PROGRAM OUTPUTS
VAR
	C6_K1_SAFETY_CONTACTOR AT %Q*: BOOL; // 
	C6_K2_SAFETY_CONTACTOR AT %Q*: BOOL; // 
	C7_K1_SAFETY_CONTACTOR AT %Q*: BOOL; // 
	C7_K2_SAFETY_CONTACTOR AT %Q*: BOOL; // 	



KIRK_BIT: BOOL;
BTEST :BOOL;
	
//GL4: sConveyor;
	

//GL5A:sConveyor;
	
	
//GL5B: sConveyor;
//GL6: sConveyor;
//GL7: sConveyor;
//GL8: sConveyor;
//GL9: sConveyor;
	
END_VAR

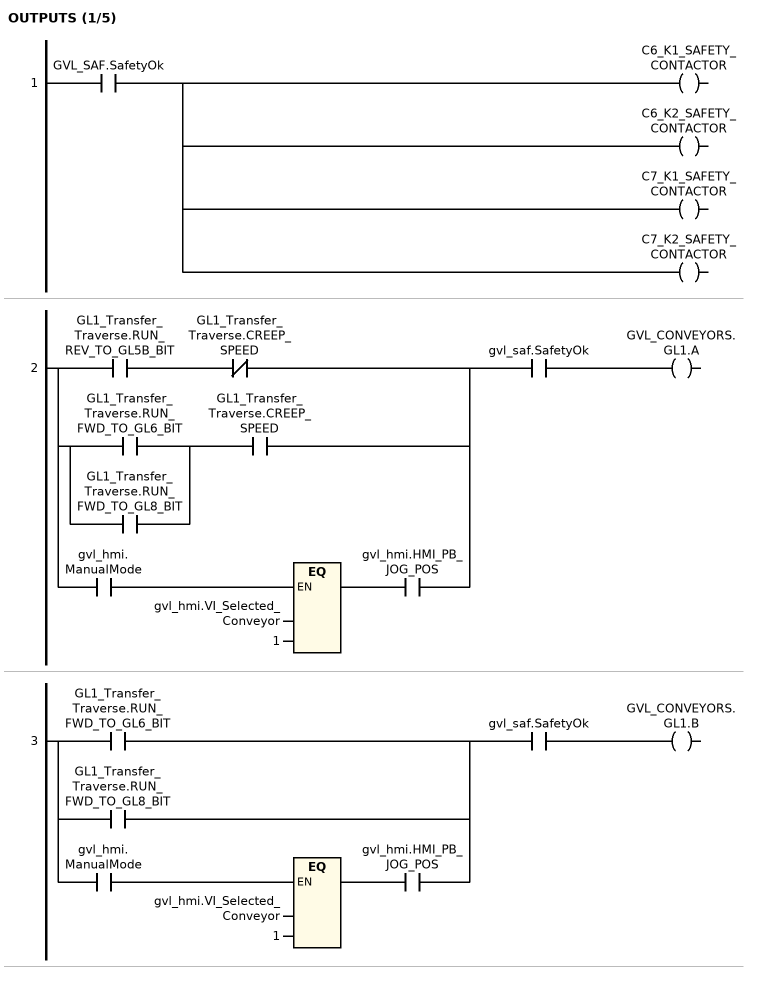
// NETWORK 1
C6_K1_SAFETY_CONTACTOR := GVL_SAF.SafetyOk;
C6_K2_SAFETY_CONTACTOR := GVL_SAF.SafetyOk;
C7_K1_SAFETY_CONTACTOR := GVL_SAF.SafetyOk;
C7_K2_SAFETY_CONTACTOR := GVL_SAF.SafetyOk;

// NETWORK 2
GVL_CONVEYORS.GL1.A := (GL1_Transfer_Traverse.RUN_REV_TO_GL5B_BIT AND NOT GL1_Transfer_Traverse.CREEP_SPEED OR (GL1_Transfer_Traverse.RUN_FWD_TO_GL6_BIT OR GL1_Transfer_Traverse.RUN_FWD_TO_GL8_BIT) AND GL1_Transfer_Traverse.CREEP_SPEED OR (gvl_hmi.ManualMode AND gvl_hmi.VI_Selected_Conveyor = 1) AND gvl_hmi.HMI_PB_JOG_POS) AND gvl_saf.SafetyOk;

// NETWORK 3
GVL_CONVEYORS.GL1.B := (GL1_Transfer_Traverse.RUN_FWD_TO_GL6_BIT OR GL1_Transfer_Traverse.RUN_FWD_TO_GL8_BIT OR (gvl_hmi.ManualMode AND gvl_hmi.VI_Selected_Conveyor = 1) AND gvl_hmi.HMI_PB_JOG_POS) AND gvl_saf.SafetyOk;

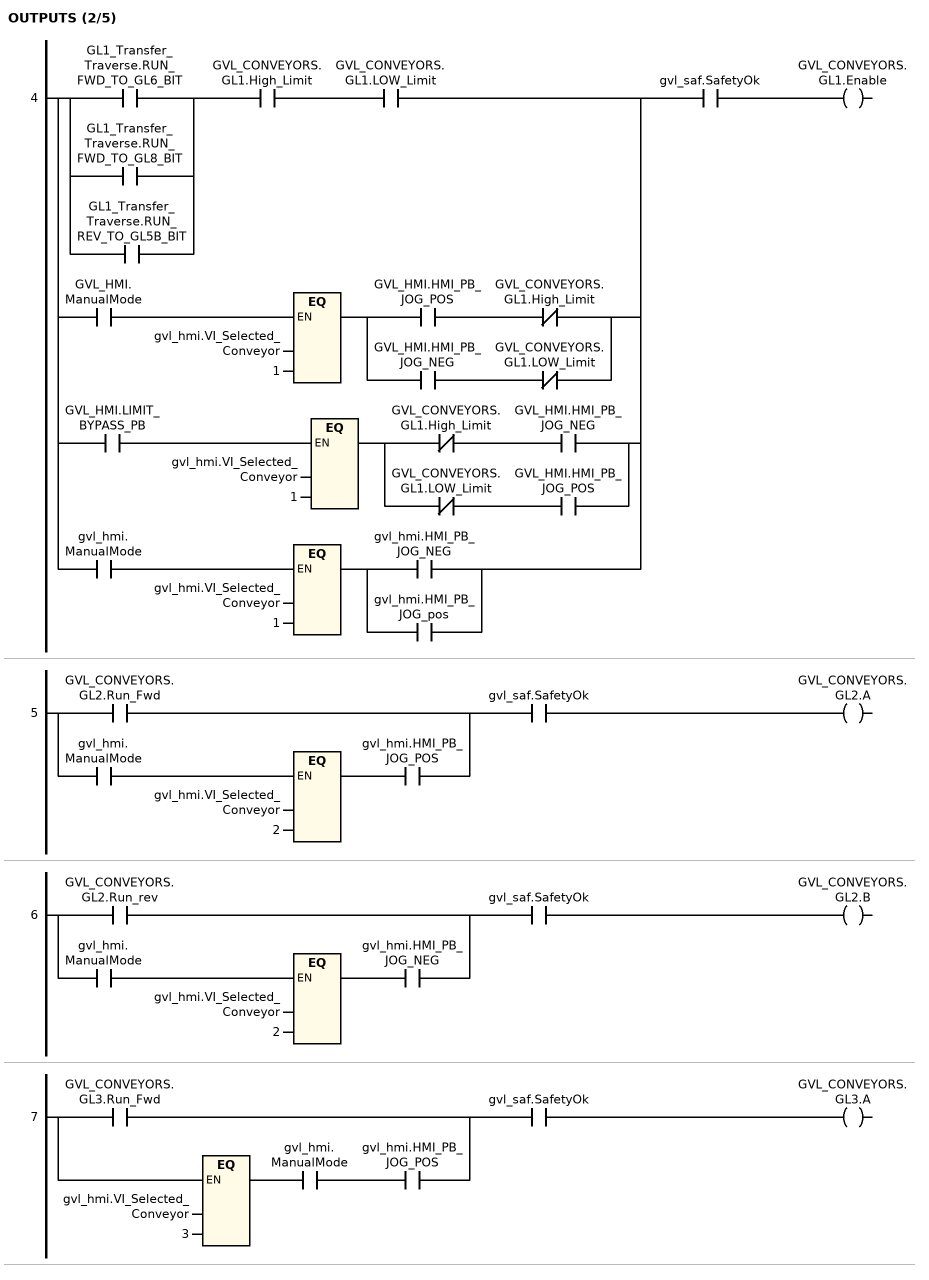
// NETWORK 4
GVL_CONVEYORS.GL1.Enable := ((GL1_Transfer_Traverse.RUN_FWD_TO_GL6_BIT OR GL1_Transfer_Traverse.RUN_FWD_TO_GL8_BIT OR GL1_Transfer_Traverse.RUN_REV_TO_GL5B_BIT) AND GVL_CONVEYORS.GL1.High_Limit AND GVL_CONVEYORS.GL1.LOW_Limit OR (GVL_HMI.ManualMode AND gvl_hmi.VI_Selected_Conveyor = 1) AND (GVL_HMI.HMI_PB_JOG_POS AND NOT GVL_CONVEYORS.GL1.High_Limit OR GVL_HMI.HMI_PB_JOG_NEG AND NOT GVL_CONVEYORS.GL1.LOW_Limit) OR (GVL_HMI.LIMIT_BYPASS_PB AND gvl_hmi.VI_Selected_Conveyor = 1) AND (NOT GVL_CONVEYORS.GL1.High_Limit AND GVL_HMI.HMI_PB_JOG_NEG OR NOT GVL_CONVEYORS.GL1.LOW_Limit AND GVL_HMI.HMI_PB_JOG_POS) OR (gvl_hmi.ManualMode AND gvl_hmi.VI_Selected_Conveyor = 1) AND (gvl_hmi.HMI_PB_JOG_NEG OR gvl_hmi.HMI_PB_JOG_pos)) AND gvl_saf.SafetyOk;

// NETWORK 5
GVL_CONVEYORS.GL2.A := (GVL_CONVEYORS.GL2.Run_Fwd OR (gvl_hmi.ManualMode AND gvl_hmi.VI_Selected_Conveyor = 2) AND gvl_hmi.HMI_PB_JOG_POS) AND gvl_saf.SafetyOk;

// NETWORK 6
GVL_CONVEYORS.GL2.B := (GVL_CONVEYORS.GL2.Run_rev OR (gvl_hmi.ManualMode AND gvl_hmi.VI_Selected_Conveyor = 2) AND gvl_hmi.HMI_PB_JOG_NEG) AND gvl_saf.SafetyOk;

// NETWORK 7
GVL_CONVEYORS.GL3.A := (GVL_CONVEYORS.GL3.Run_Fwd OR gvl_hmi.VI_Selected_Conveyor = 3 AND gvl_hmi.ManualMode AND gvl_hmi.HMI_PB_JOG_POS) AND gvl_saf.SafetyOk;

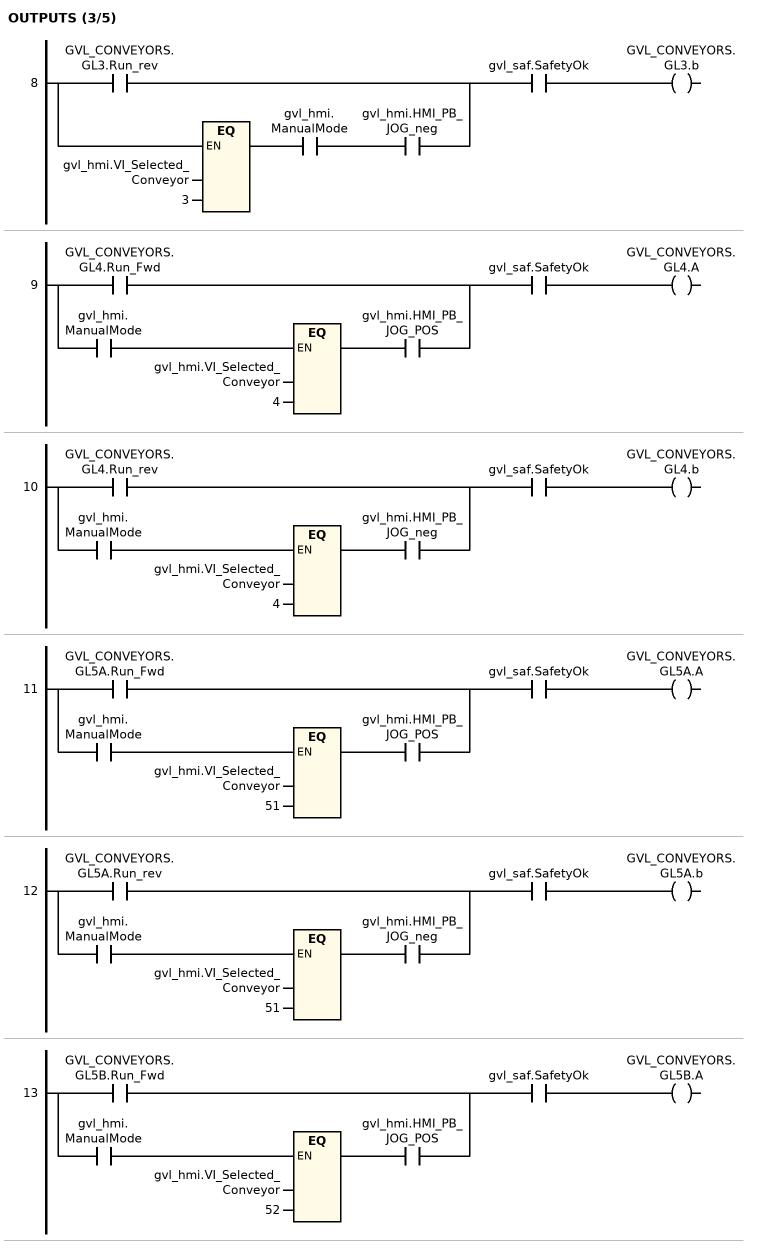
// NETWORK 8
GVL_CONVEYORS.GL3.b := (GVL_CONVEYORS.GL3.Run_rev OR gvl_hmi.VI_Selected_Conveyor = 3 AND gvl_hmi.ManualMode AND gvl_hmi.HMI_PB_JOG_neg) AND gvl_saf.SafetyOk;

// NETWORK 9
GVL_CONVEYORS.GL4.A := (GVL_CONVEYORS.GL4.Run_Fwd OR (gvl_hmi.ManualMode AND gvl_hmi.VI_Selected_Conveyor = 4) AND gvl_hmi.HMI_PB_JOG_POS) AND gvl_saf.SafetyOk;

// NETWORK 10
GVL_CONVEYORS.GL4.b := (GVL_CONVEYORS.GL4.Run_rev OR (gvl_hmi.ManualMode AND gvl_hmi.VI_Selected_Conveyor = 4) AND gvl_hmi.HMI_PB_JOG_neg) AND gvl_saf.SafetyOk;

// NETWORK 11
GVL_CONVEYORS.GL5A.A := (GVL_CONVEYORS.GL5A.Run_Fwd OR (gvl_hmi.ManualMode AND gvl_hmi.VI_Selected_Conveyor = 51) AND gvl_hmi.HMI_PB_JOG_POS) AND gvl_saf.SafetyOk;

// NETWORK 12
GVL_CONVEYORS.GL5A.b := (GVL_CONVEYORS.GL5A.Run_rev OR (gvl_hmi.ManualMode AND gvl_hmi.VI_Selected_Conveyor = 51) AND gvl_hmi.HMI_PB_JOG_neg) AND gvl_saf.SafetyOk;

// NETWORK 13
GVL_CONVEYORS.GL5B.A := (GVL_CONVEYORS.GL5B.Run_Fwd OR (gvl_hmi.ManualMode AND gvl_hmi.VI_Selected_Conveyor = 52) AND gvl_hmi.HMI_PB_JOG_POS) AND gvl_saf.SafetyOk;

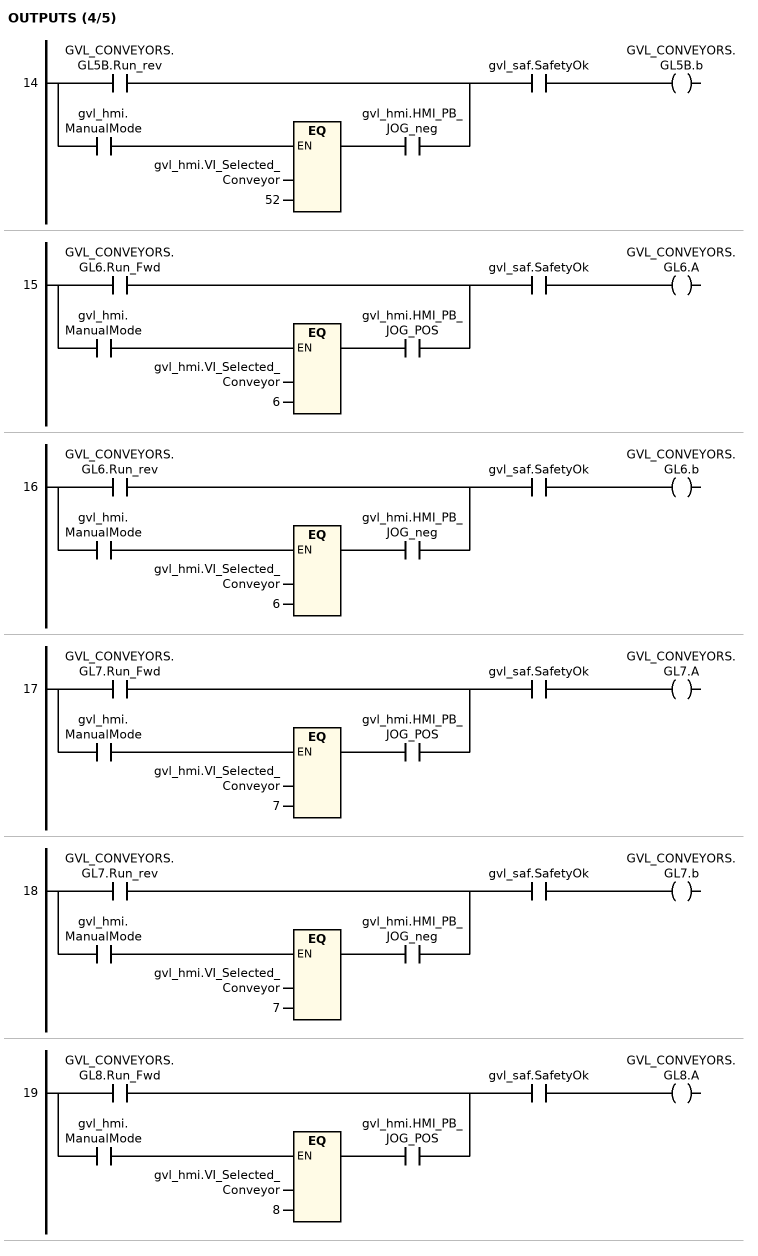
// NETWORK 14
GVL_CONVEYORS.GL5B.b := (GVL_CONVEYORS.GL5B.Run_rev OR (gvl_hmi.ManualMode AND gvl_hmi.VI_Selected_Conveyor = 52) AND gvl_hmi.HMI_PB_JOG_neg) AND gvl_saf.SafetyOk;

// NETWORK 15
GVL_CONVEYORS.GL6.A := (GVL_CONVEYORS.GL6.Run_Fwd OR (gvl_hmi.ManualMode AND gvl_hmi.VI_Selected_Conveyor = 6) AND gvl_hmi.HMI_PB_JOG_POS) AND gvl_saf.SafetyOk;

// NETWORK 16
GVL_CONVEYORS.GL6.b := (GVL_CONVEYORS.GL6.Run_rev OR (gvl_hmi.ManualMode AND gvl_hmi.VI_Selected_Conveyor = 6) AND gvl_hmi.HMI_PB_JOG_neg) AND gvl_saf.SafetyOk;

// NETWORK 17
GVL_CONVEYORS.GL7.A := (GVL_CONVEYORS.GL7.Run_Fwd OR (gvl_hmi.ManualMode AND gvl_hmi.VI_Selected_Conveyor = 7) AND gvl_hmi.HMI_PB_JOG_POS) AND gvl_saf.SafetyOk;

// NETWORK 18
GVL_CONVEYORS.GL7.b := (GVL_CONVEYORS.GL7.Run_rev OR (gvl_hmi.ManualMode AND gvl_hmi.VI_Selected_Conveyor = 7) AND gvl_hmi.HMI_PB_JOG_neg) AND gvl_saf.SafetyOk;

// NETWORK 19
GVL_CONVEYORS.GL8.A := (GVL_CONVEYORS.GL8.Run_Fwd OR (gvl_hmi.ManualMode AND gvl_hmi.VI_Selected_Conveyor = 8) AND gvl_hmi.HMI_PB_JOG_POS) AND gvl_saf.SafetyOk;

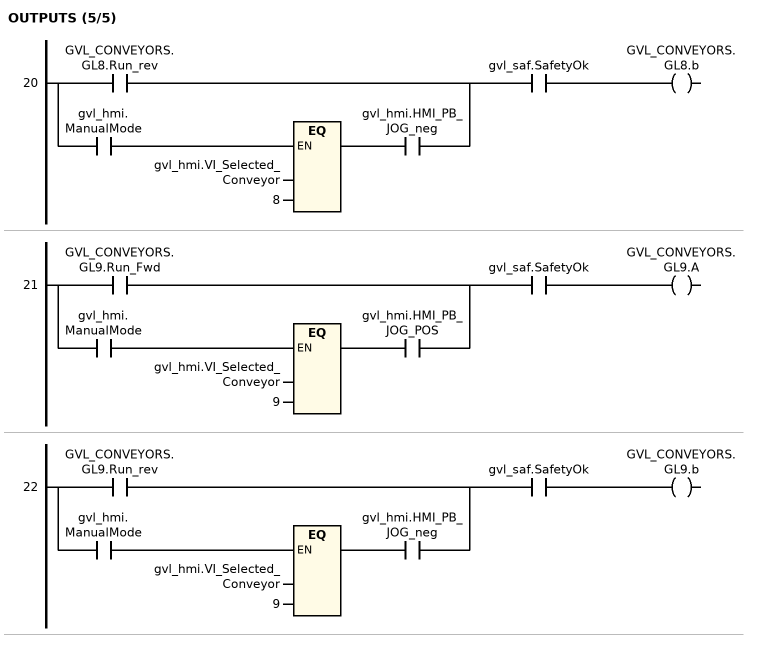
// NETWORK 20
GVL_CONVEYORS.GL8.b := (GVL_CONVEYORS.GL8.Run_rev OR (gvl_hmi.ManualMode AND gvl_hmi.VI_Selected_Conveyor = 8) AND gvl_hmi.HMI_PB_JOG_neg) AND gvl_saf.SafetyOk;

// NETWORK 21
GVL_CONVEYORS.GL9.A := (GVL_CONVEYORS.GL9.Run_Fwd OR (gvl_hmi.ManualMode AND gvl_hmi.VI_Selected_Conveyor = 9) AND gvl_hmi.HMI_PB_JOG_POS) AND gvl_saf.SafetyOk;

// NETWORK 22
GVL_CONVEYORS.GL9.b := (GVL_CONVEYORS.GL9.Run_rev OR (gvl_hmi.ManualMode AND gvl_hmi.VI_Selected_Conveyor = 9) AND gvl_hmi.HMI_PB_JOG_neg) AND gvl_saf.SafetyOk;

END_PROGRAM

(* stored: Version 1.1.0.1, ProductVersion 3.1.4024.12
   POU OUTPUTS: Id {b8a21824-47d8-40ce-a09e-f966e96d1f20}, SpecialFunc None *)
